// TIA Portal V17 export
// export: Created 2025-07-01T09:58:25.4469357Z, ExportSetting WithDefaults, DisplayName Totally Integrated Automation Portal, DisplayVersion V17 Update 8, DisplayName TIA Portal Openness, DisplayVersion V17 Update 8, DisplayName TIA Portal Version Control Interface, DisplayVersion V17, DisplayName SINAMICS Startdrive Advanced, DisplayVersion V17 SP2, DisplayName SINAMICS Startdrive G110M, G120, G120C, G120D, G120P, G115D, DisplayVersion V17 SP2, DisplayName SINAMICS Startdrive G130, G150, S120, S150, SINAMICS MV, S210, DisplayVersion V17 SP2, DisplayName STEP 7 Professional, DisplayVersion V17 Update 8, DisplayName SINUMERIK ONE STEP 7 Toolbox, DisplayVersion V17 Update 12, DisplayName SINUMERIK ONE PLC Basic Program Plus, DisplayVersion V17 Update 12, DisplayName SINUMERIK 840D sl STEP 7 Toolbox, DisplayVersion V17 Update 12, DisplayName STEP 7 Safety, DisplayVersion V17 Update 6, DisplayName WinCC Advanced, DisplayVersion V17 Update 8
FUNCTION "FC2500_UNIT_1_FIXTURES" : Void   // FC2500, LAD
TITLE = FIXTURE 1
{ S7_Optimized_Access := 'FALSE' }
AUTHOR : ETXETAR
VERSION : 1.0
// stored: AutoNumber false, IsIECCheckEnabled false, SetENOAutomatically false, UDAEnableTagReadback false
   VAR CONSTANT
      FC_NUMBER : DInt := 2500;
   END_VAR
BEGIN

REGION Network 1: CALL FB2500 FIXTURE 1 UNIT 1 CLADDING
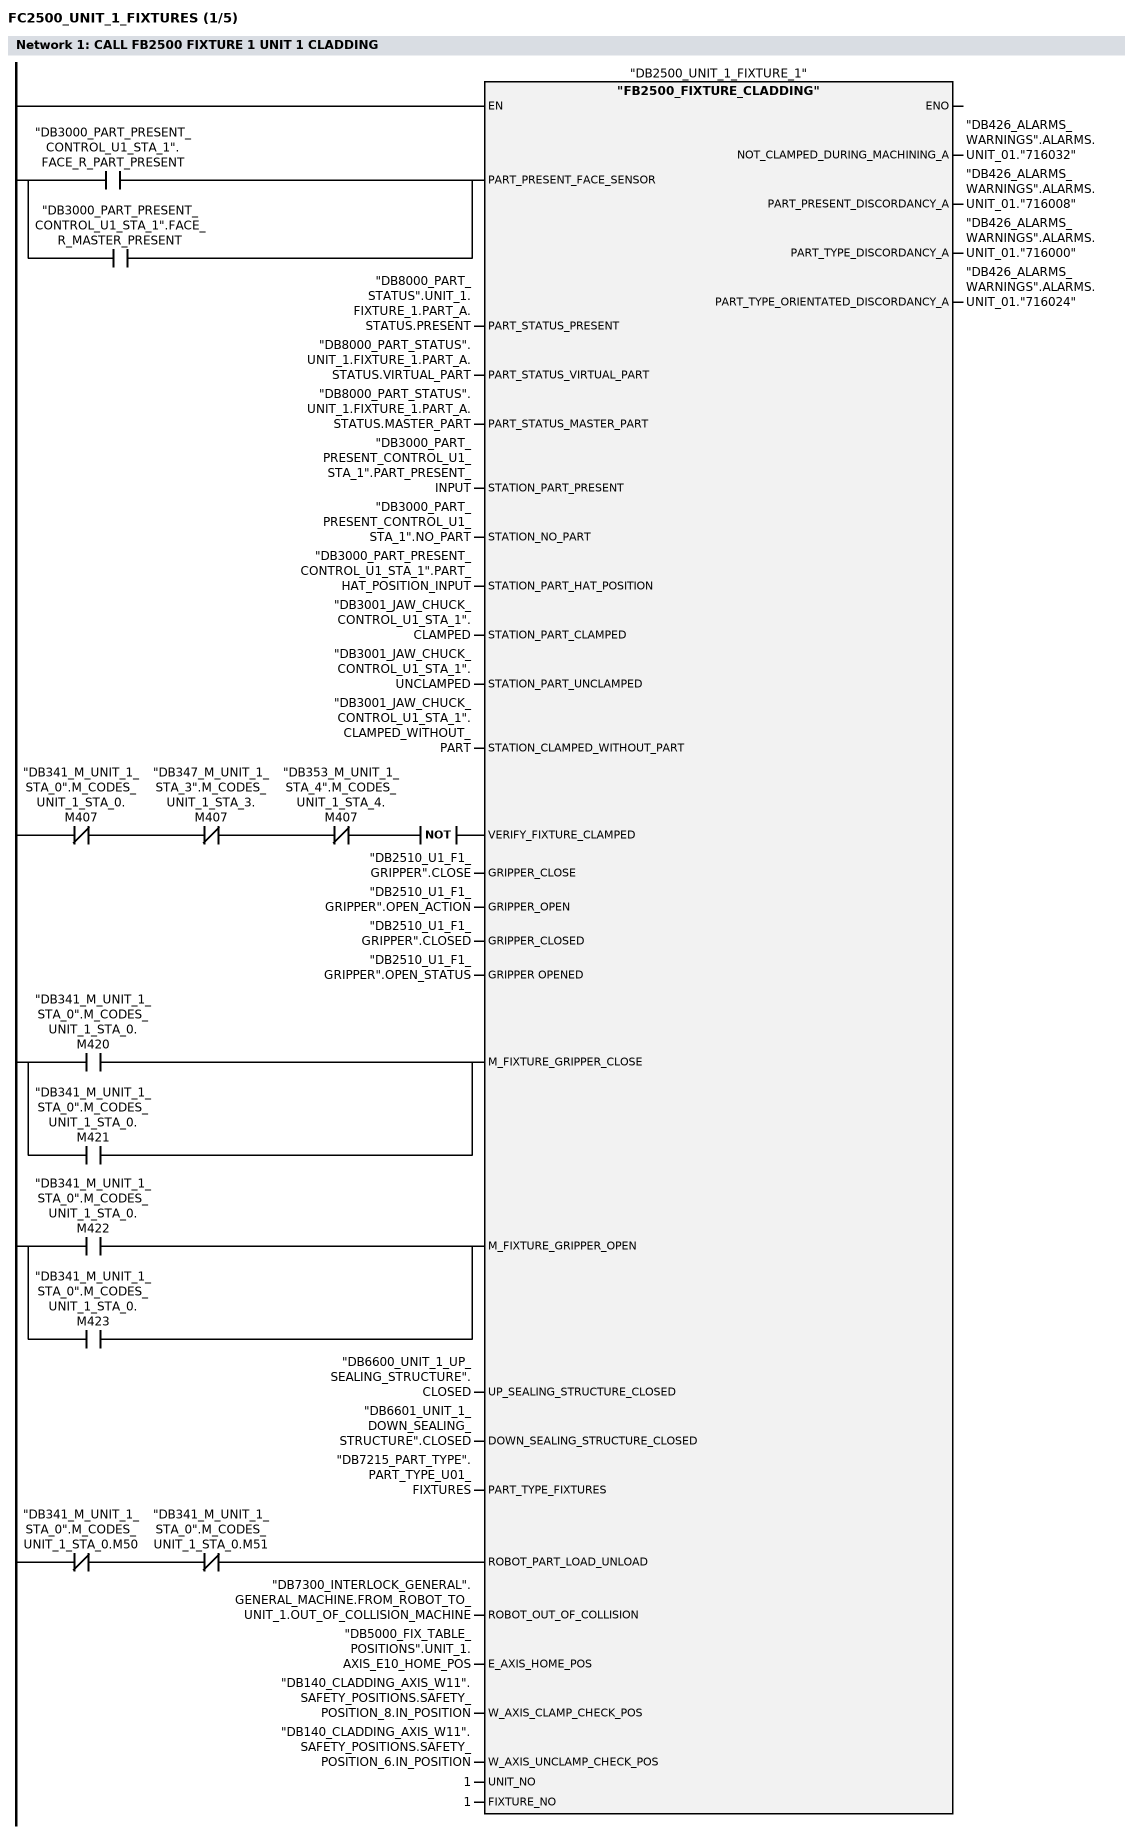
   RUNG wire#powerrail
      "DB2500_UNIT_1_FIXTURE_1"(PART_PRESENT_FACE_SENSOR := wire#w1, VERIFY_FIXTURE_CLAMPED := wire#w2, M_FIXTURE_GRIPPER_CLOSE := wire#w3, M_FIXTURE_GRIPPER_OPEN := wire#w4, ROBOT_PART_LOAD_UNLOAD := wire#w5, PART_STATUS_PRESENT := "DB8000_PART_STATUS".UNIT_1.FIXTURE_1.PART_A.STATUS.PRESENT, PART_STATUS_VIRTUAL_PART := "DB8000_PART_STATUS".UNIT_1.FIXTURE_1.PART_A.STATUS.VIRTUAL_PART, PART_STATUS_MASTER_PART := "DB8000_PART_STATUS".UNIT_1.FIXTURE_1.PART_A.STATUS.MASTER_PART, STATION_PART_PRESENT := "DB3000_PART_PRESENT_CONTROL_U1_STA_1".PART_PRESENT_INPUT, STATION_NO_PART := "DB3000_PART_PRESENT_CONTROL_U1_STA_1".NO_PART, STATION_PART_HAT_POSITION := "DB3000_PART_PRESENT_CONTROL_U1_STA_1".PART_HAT_POSITION_INPUT, STATION_PART_CLAMPED := "DB3001_JAW_CHUCK_CONTROL_U1_STA_1".CLAMPED, STATION_PART_UNCLAMPED := "DB3001_JAW_CHUCK_CONTROL_U1_STA_1".UNCLAMPED, STATION_CLAMPED_WITHOUT_PART := "DB3001_JAW_CHUCK_CONTROL_U1_STA_1".CLAMPED_WITHOUT_PART, GRIPPER_CLOSE := "DB2510_U1_F1_GRIPPER".CLOSE, GRIPPER_OPEN := "DB2510_U1_F1_GRIPPER".OPEN_ACTION, GRIPPER_CLOSED := "DB2510_U1_F1_GRIPPER".CLOSED, "GRIPPER OPENED" := "DB2510_U1_F1_GRIPPER".OPEN_STATUS, UP_SEALING_STRUCTURE_CLOSED := "DB6600_UNIT_1_UP_SEALING_STRUCTURE".CLOSED, DOWN_SEALING_STRUCTURE_CLOSED := "DB6601_UNIT_1_DOWN_SEALING_STRUCTURE".CLOSED, PART_TYPE_FIXTURES := "DB7215_PART_TYPE".PART_TYPE_U01_FIXTURES, ROBOT_OUT_OF_COLLISION := "DB7300_INTERLOCK_GENERAL".GENERAL_MACHINE.FROM_ROBOT_TO_UNIT_1.OUT_OF_COLLISION_MACHINE, E_AXIS_HOME_POS := "DB5000_FIX_TABLE_POSITIONS".UNIT_1.AXIS_E10_HOME_POS, W_AXIS_CLAMP_CHECK_POS := "DB140_CLADDING_AXIS_W11".SAFETY_POSITIONS.SAFETY_POSITION_8.IN_POSITION, W_AXIS_UNCLAMP_CHECK_POS := "DB140_CLADDING_AXIS_W11".SAFETY_POSITIONS.SAFETY_POSITION_6.IN_POSITION, UNIT_NO := 1, FIXTURE_NO := 1, NOT_CLAMPED_DURING_MACHINING_A => "DB426_ALARMS_WARNINGS".ALARMS.UNIT_01."716032", PART_PRESENT_DISCORDANCY_A => "DB426_ALARMS_WARNINGS".ALARMS.UNIT_01."716008", PART_TYPE_DISCORDANCY_A => "DB426_ALARMS_WARNINGS".ALARMS.UNIT_01."716000", PART_TYPE_ORIENTATED_DISCORDANCY_A => "DB426_ALARMS_WARNINGS".ALARMS.UNIT_01."716024")
   END_RUNG
   RUNG wire#powerrail
      Contact( "DB3000_PART_PRESENT_CONTROL_U1_STA_1".FACE_R_PART_PRESENT )
   END_RUNG wire#w1
   RUNG wire#powerrail
      Contact( "DB3000_PART_PRESENT_CONTROL_U1_STA_1".FACE_R_MASTER_PRESENT )
   END_RUNG wire#w1
   RUNG wire#powerrail
      I_Contact( "DB341_M_UNIT_1_STA_0".M_CODES_UNIT_1_STA_0.M407 )
      I_Contact( "DB347_M_UNIT_1_STA_3".M_CODES_UNIT_1_STA_3.M407 )
      I_Contact( "DB353_M_UNIT_1_STA_4".M_CODES_UNIT_1_STA_4.M407 )
      Not()
   END_RUNG wire#w2
   RUNG wire#powerrail
      Contact( "DB341_M_UNIT_1_STA_0".M_CODES_UNIT_1_STA_0.M420 )
   END_RUNG wire#w3
   RUNG wire#powerrail
      Contact( "DB341_M_UNIT_1_STA_0".M_CODES_UNIT_1_STA_0.M421 )
   END_RUNG wire#w3
   RUNG wire#powerrail
      Contact( "DB341_M_UNIT_1_STA_0".M_CODES_UNIT_1_STA_0.M422 )
   END_RUNG wire#w4
   RUNG wire#powerrail
      Contact( "DB341_M_UNIT_1_STA_0".M_CODES_UNIT_1_STA_0.M423 )
   END_RUNG wire#w4
   RUNG wire#powerrail
      I_Contact( "DB341_M_UNIT_1_STA_0".M_CODES_UNIT_1_STA_0.M50 )
      I_Contact( "DB341_M_UNIT_1_STA_0".M_CODES_UNIT_1_STA_0.M51 )
   END_RUNG wire#w5
   // the same network as SCL:
   "DB2500_UNIT_1_FIXTURE_1"(PART_PRESENT_FACE_SENSOR := "DB3000_PART_PRESENT_CONTROL_U1_STA_1".FACE_R_PART_PRESENT OR "DB3000_PART_PRESENT_CONTROL_U1_STA_1".FACE_R_MASTER_PRESENT,   // "FB2500_FIXTURE_CLADDING"
                           PART_STATUS_PRESENT := "DB8000_PART_STATUS".UNIT_1.FIXTURE_1.PART_A.STATUS.PRESENT,
                           PART_STATUS_VIRTUAL_PART := "DB8000_PART_STATUS".UNIT_1.FIXTURE_1.PART_A.STATUS.VIRTUAL_PART,
                           PART_STATUS_MASTER_PART := "DB8000_PART_STATUS".UNIT_1.FIXTURE_1.PART_A.STATUS.MASTER_PART,
                           STATION_PART_PRESENT := "DB3000_PART_PRESENT_CONTROL_U1_STA_1".PART_PRESENT_INPUT,
                           STATION_NO_PART := "DB3000_PART_PRESENT_CONTROL_U1_STA_1".NO_PART,
                           STATION_PART_HAT_POSITION := "DB3000_PART_PRESENT_CONTROL_U1_STA_1".PART_HAT_POSITION_INPUT,
                           STATION_PART_CLAMPED := "DB3001_JAW_CHUCK_CONTROL_U1_STA_1".CLAMPED,
                           STATION_PART_UNCLAMPED := "DB3001_JAW_CHUCK_CONTROL_U1_STA_1".UNCLAMPED,
                           STATION_CLAMPED_WITHOUT_PART := "DB3001_JAW_CHUCK_CONTROL_U1_STA_1".CLAMPED_WITHOUT_PART,
                           VERIFY_FIXTURE_CLAMPED := NOT (NOT "DB341_M_UNIT_1_STA_0".M_CODES_UNIT_1_STA_0.M407 AND NOT "DB347_M_UNIT_1_STA_3".M_CODES_UNIT_1_STA_3.M407 AND NOT "DB353_M_UNIT_1_STA_4".M_CODES_UNIT_1_STA_4.M407),
                           GRIPPER_CLOSE := "DB2510_U1_F1_GRIPPER".CLOSE,
                           GRIPPER_OPEN := "DB2510_U1_F1_GRIPPER".OPEN_ACTION,
                           GRIPPER_CLOSED := "DB2510_U1_F1_GRIPPER".CLOSED,
                           "GRIPPER OPENED" := "DB2510_U1_F1_GRIPPER".OPEN_STATUS,
                           M_FIXTURE_GRIPPER_CLOSE := "DB341_M_UNIT_1_STA_0".M_CODES_UNIT_1_STA_0.M420 OR "DB341_M_UNIT_1_STA_0".M_CODES_UNIT_1_STA_0.M421,
                           M_FIXTURE_GRIPPER_OPEN := "DB341_M_UNIT_1_STA_0".M_CODES_UNIT_1_STA_0.M422 OR "DB341_M_UNIT_1_STA_0".M_CODES_UNIT_1_STA_0.M423,
                           UP_SEALING_STRUCTURE_CLOSED := "DB6600_UNIT_1_UP_SEALING_STRUCTURE".CLOSED,
                           DOWN_SEALING_STRUCTURE_CLOSED := "DB6601_UNIT_1_DOWN_SEALING_STRUCTURE".CLOSED,
                           PART_TYPE_FIXTURES := "DB7215_PART_TYPE".PART_TYPE_U01_FIXTURES,
                           ROBOT_PART_LOAD_UNLOAD := NOT "DB341_M_UNIT_1_STA_0".M_CODES_UNIT_1_STA_0.M50 AND NOT "DB341_M_UNIT_1_STA_0".M_CODES_UNIT_1_STA_0.M51,
                           ROBOT_OUT_OF_COLLISION := "DB7300_INTERLOCK_GENERAL".GENERAL_MACHINE.FROM_ROBOT_TO_UNIT_1.OUT_OF_COLLISION_MACHINE,
                           E_AXIS_HOME_POS := "DB5000_FIX_TABLE_POSITIONS".UNIT_1.AXIS_E10_HOME_POS,
                           W_AXIS_CLAMP_CHECK_POS := "DB140_CLADDING_AXIS_W11".SAFETY_POSITIONS.SAFETY_POSITION_8.IN_POSITION,
                           W_AXIS_UNCLAMP_CHECK_POS := "DB140_CLADDING_AXIS_W11".SAFETY_POSITIONS.SAFETY_POSITION_6.IN_POSITION,
                           UNIT_NO := 1,
                           FIXTURE_NO := 1,
                           NOT_CLAMPED_DURING_MACHINING_A => "DB426_ALARMS_WARNINGS".ALARMS.UNIT_01."716032",
                           PART_PRESENT_DISCORDANCY_A => "DB426_ALARMS_WARNINGS".ALARMS.UNIT_01."716008",
                           PART_TYPE_DISCORDANCY_A => "DB426_ALARMS_WARNINGS".ALARMS.UNIT_01."716000",
                           PART_TYPE_ORIENTATED_DISCORDANCY_A => "DB426_ALARMS_WARNINGS".ALARMS.UNIT_01."716024");
END_REGION

REGION Network 2: CALL FB2600 FIXTURE 2 UNIT 1 CLADDING
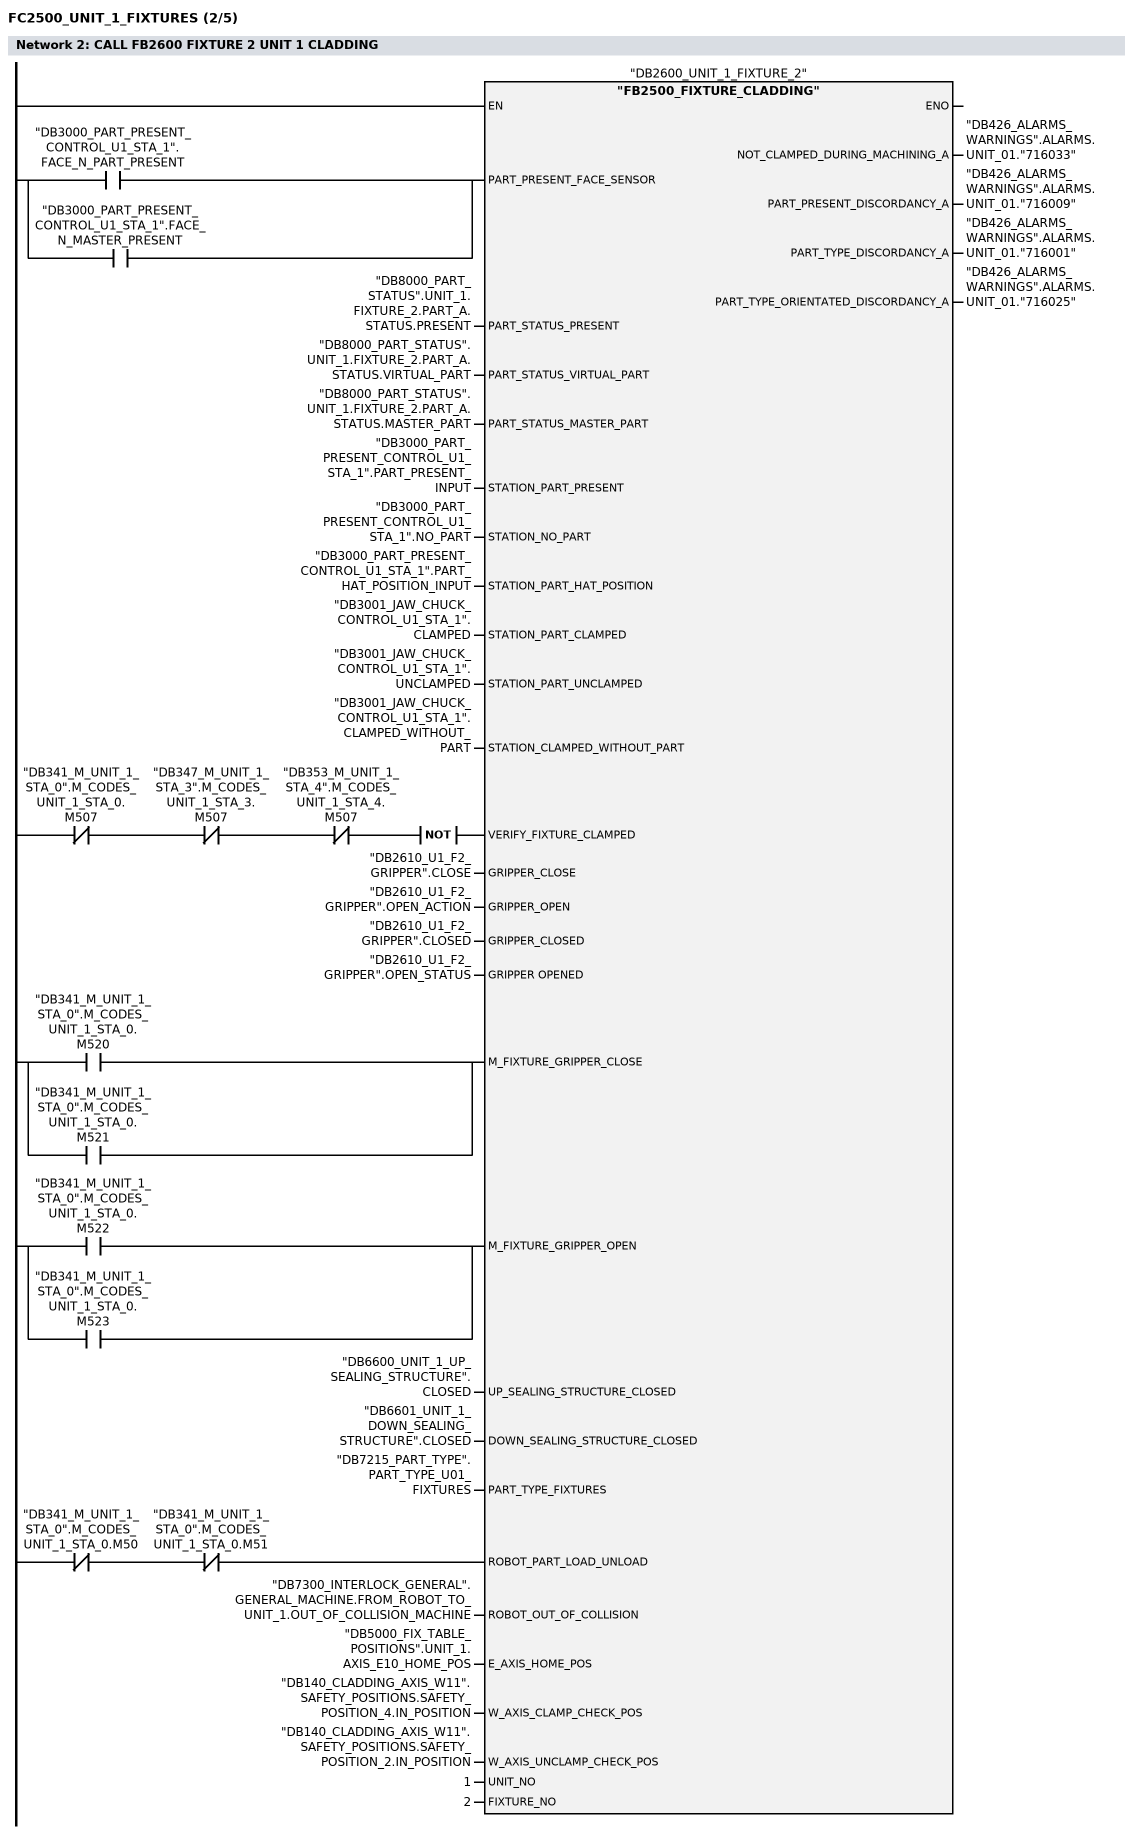
   RUNG wire#powerrail
      "DB2600_UNIT_1_FIXTURE_2"(PART_PRESENT_FACE_SENSOR := wire#w1, VERIFY_FIXTURE_CLAMPED := wire#w2, M_FIXTURE_GRIPPER_CLOSE := wire#w3, M_FIXTURE_GRIPPER_OPEN := wire#w4, ROBOT_PART_LOAD_UNLOAD := wire#w5, PART_STATUS_PRESENT := "DB8000_PART_STATUS".UNIT_1.FIXTURE_2.PART_A.STATUS.PRESENT, PART_STATUS_VIRTUAL_PART := "DB8000_PART_STATUS".UNIT_1.FIXTURE_2.PART_A.STATUS.VIRTUAL_PART, PART_STATUS_MASTER_PART := "DB8000_PART_STATUS".UNIT_1.FIXTURE_2.PART_A.STATUS.MASTER_PART, STATION_PART_PRESENT := "DB3000_PART_PRESENT_CONTROL_U1_STA_1".PART_PRESENT_INPUT, STATION_NO_PART := "DB3000_PART_PRESENT_CONTROL_U1_STA_1".NO_PART, STATION_PART_HAT_POSITION := "DB3000_PART_PRESENT_CONTROL_U1_STA_1".PART_HAT_POSITION_INPUT, STATION_PART_CLAMPED := "DB3001_JAW_CHUCK_CONTROL_U1_STA_1".CLAMPED, STATION_PART_UNCLAMPED := "DB3001_JAW_CHUCK_CONTROL_U1_STA_1".UNCLAMPED, STATION_CLAMPED_WITHOUT_PART := "DB3001_JAW_CHUCK_CONTROL_U1_STA_1".CLAMPED_WITHOUT_PART, GRIPPER_CLOSE := "DB2610_U1_F2_GRIPPER".CLOSE, GRIPPER_OPEN := "DB2610_U1_F2_GRIPPER".OPEN_ACTION, GRIPPER_CLOSED := "DB2610_U1_F2_GRIPPER".CLOSED, "GRIPPER OPENED" := "DB2610_U1_F2_GRIPPER".OPEN_STATUS, UP_SEALING_STRUCTURE_CLOSED := "DB6600_UNIT_1_UP_SEALING_STRUCTURE".CLOSED, DOWN_SEALING_STRUCTURE_CLOSED := "DB6601_UNIT_1_DOWN_SEALING_STRUCTURE".CLOSED, PART_TYPE_FIXTURES := "DB7215_PART_TYPE".PART_TYPE_U01_FIXTURES, ROBOT_OUT_OF_COLLISION := "DB7300_INTERLOCK_GENERAL".GENERAL_MACHINE.FROM_ROBOT_TO_UNIT_1.OUT_OF_COLLISION_MACHINE, E_AXIS_HOME_POS := "DB5000_FIX_TABLE_POSITIONS".UNIT_1.AXIS_E10_HOME_POS, W_AXIS_CLAMP_CHECK_POS := "DB140_CLADDING_AXIS_W11".SAFETY_POSITIONS.SAFETY_POSITION_4.IN_POSITION, W_AXIS_UNCLAMP_CHECK_POS := "DB140_CLADDING_AXIS_W11".SAFETY_POSITIONS.SAFETY_POSITION_2.IN_POSITION, UNIT_NO := 1, FIXTURE_NO := 2, NOT_CLAMPED_DURING_MACHINING_A => "DB426_ALARMS_WARNINGS".ALARMS.UNIT_01."716033", PART_PRESENT_DISCORDANCY_A => "DB426_ALARMS_WARNINGS".ALARMS.UNIT_01."716009", PART_TYPE_DISCORDANCY_A => "DB426_ALARMS_WARNINGS".ALARMS.UNIT_01."716001", PART_TYPE_ORIENTATED_DISCORDANCY_A => "DB426_ALARMS_WARNINGS".ALARMS.UNIT_01."716025")
   END_RUNG
   RUNG wire#powerrail
      Contact( "DB3000_PART_PRESENT_CONTROL_U1_STA_1".FACE_N_PART_PRESENT )
   END_RUNG wire#w1
   RUNG wire#powerrail
      Contact( "DB3000_PART_PRESENT_CONTROL_U1_STA_1".FACE_N_MASTER_PRESENT )
   END_RUNG wire#w1
   RUNG wire#powerrail
      I_Contact( "DB341_M_UNIT_1_STA_0".M_CODES_UNIT_1_STA_0.M507 )
      I_Contact( "DB347_M_UNIT_1_STA_3".M_CODES_UNIT_1_STA_3.M507 )
      I_Contact( "DB353_M_UNIT_1_STA_4".M_CODES_UNIT_1_STA_4.M507 )
      Not()
   END_RUNG wire#w2
   RUNG wire#powerrail
      Contact( "DB341_M_UNIT_1_STA_0".M_CODES_UNIT_1_STA_0.M520 )
   END_RUNG wire#w3
   RUNG wire#powerrail
      Contact( "DB341_M_UNIT_1_STA_0".M_CODES_UNIT_1_STA_0.M521 )
   END_RUNG wire#w3
   RUNG wire#powerrail
      Contact( "DB341_M_UNIT_1_STA_0".M_CODES_UNIT_1_STA_0.M522 )
   END_RUNG wire#w4
   RUNG wire#powerrail
      Contact( "DB341_M_UNIT_1_STA_0".M_CODES_UNIT_1_STA_0.M523 )
   END_RUNG wire#w4
   RUNG wire#powerrail
      I_Contact( "DB341_M_UNIT_1_STA_0".M_CODES_UNIT_1_STA_0.M50 )
      I_Contact( "DB341_M_UNIT_1_STA_0".M_CODES_UNIT_1_STA_0.M51 )
   END_RUNG wire#w5
   // the same network as SCL:
   "DB2600_UNIT_1_FIXTURE_2"(PART_PRESENT_FACE_SENSOR := "DB3000_PART_PRESENT_CONTROL_U1_STA_1".FACE_N_PART_PRESENT OR "DB3000_PART_PRESENT_CONTROL_U1_STA_1".FACE_N_MASTER_PRESENT,   // "FB2500_FIXTURE_CLADDING"
                           PART_STATUS_PRESENT := "DB8000_PART_STATUS".UNIT_1.FIXTURE_2.PART_A.STATUS.PRESENT,
                           PART_STATUS_VIRTUAL_PART := "DB8000_PART_STATUS".UNIT_1.FIXTURE_2.PART_A.STATUS.VIRTUAL_PART,
                           PART_STATUS_MASTER_PART := "DB8000_PART_STATUS".UNIT_1.FIXTURE_2.PART_A.STATUS.MASTER_PART,
                           STATION_PART_PRESENT := "DB3000_PART_PRESENT_CONTROL_U1_STA_1".PART_PRESENT_INPUT,
                           STATION_NO_PART := "DB3000_PART_PRESENT_CONTROL_U1_STA_1".NO_PART,
                           STATION_PART_HAT_POSITION := "DB3000_PART_PRESENT_CONTROL_U1_STA_1".PART_HAT_POSITION_INPUT,
                           STATION_PART_CLAMPED := "DB3001_JAW_CHUCK_CONTROL_U1_STA_1".CLAMPED,
                           STATION_PART_UNCLAMPED := "DB3001_JAW_CHUCK_CONTROL_U1_STA_1".UNCLAMPED,
                           STATION_CLAMPED_WITHOUT_PART := "DB3001_JAW_CHUCK_CONTROL_U1_STA_1".CLAMPED_WITHOUT_PART,
                           VERIFY_FIXTURE_CLAMPED := NOT (NOT "DB341_M_UNIT_1_STA_0".M_CODES_UNIT_1_STA_0.M507 AND NOT "DB347_M_UNIT_1_STA_3".M_CODES_UNIT_1_STA_3.M507 AND NOT "DB353_M_UNIT_1_STA_4".M_CODES_UNIT_1_STA_4.M507),
                           GRIPPER_CLOSE := "DB2610_U1_F2_GRIPPER".CLOSE,
                           GRIPPER_OPEN := "DB2610_U1_F2_GRIPPER".OPEN_ACTION,
                           GRIPPER_CLOSED := "DB2610_U1_F2_GRIPPER".CLOSED,
                           "GRIPPER OPENED" := "DB2610_U1_F2_GRIPPER".OPEN_STATUS,
                           M_FIXTURE_GRIPPER_CLOSE := "DB341_M_UNIT_1_STA_0".M_CODES_UNIT_1_STA_0.M520 OR "DB341_M_UNIT_1_STA_0".M_CODES_UNIT_1_STA_0.M521,
                           M_FIXTURE_GRIPPER_OPEN := "DB341_M_UNIT_1_STA_0".M_CODES_UNIT_1_STA_0.M522 OR "DB341_M_UNIT_1_STA_0".M_CODES_UNIT_1_STA_0.M523,
                           UP_SEALING_STRUCTURE_CLOSED := "DB6600_UNIT_1_UP_SEALING_STRUCTURE".CLOSED,
                           DOWN_SEALING_STRUCTURE_CLOSED := "DB6601_UNIT_1_DOWN_SEALING_STRUCTURE".CLOSED,
                           PART_TYPE_FIXTURES := "DB7215_PART_TYPE".PART_TYPE_U01_FIXTURES,
                           ROBOT_PART_LOAD_UNLOAD := NOT "DB341_M_UNIT_1_STA_0".M_CODES_UNIT_1_STA_0.M50 AND NOT "DB341_M_UNIT_1_STA_0".M_CODES_UNIT_1_STA_0.M51,
                           ROBOT_OUT_OF_COLLISION := "DB7300_INTERLOCK_GENERAL".GENERAL_MACHINE.FROM_ROBOT_TO_UNIT_1.OUT_OF_COLLISION_MACHINE,
                           E_AXIS_HOME_POS := "DB5000_FIX_TABLE_POSITIONS".UNIT_1.AXIS_E10_HOME_POS,
                           W_AXIS_CLAMP_CHECK_POS := "DB140_CLADDING_AXIS_W11".SAFETY_POSITIONS.SAFETY_POSITION_4.IN_POSITION,
                           W_AXIS_UNCLAMP_CHECK_POS := "DB140_CLADDING_AXIS_W11".SAFETY_POSITIONS.SAFETY_POSITION_2.IN_POSITION,
                           UNIT_NO := 1,
                           FIXTURE_NO := 2,
                           NOT_CLAMPED_DURING_MACHINING_A => "DB426_ALARMS_WARNINGS".ALARMS.UNIT_01."716033",
                           PART_PRESENT_DISCORDANCY_A => "DB426_ALARMS_WARNINGS".ALARMS.UNIT_01."716009",
                           PART_TYPE_DISCORDANCY_A => "DB426_ALARMS_WARNINGS".ALARMS.UNIT_01."716001",
                           PART_TYPE_ORIENTATED_DISCORDANCY_A => "DB426_ALARMS_WARNINGS".ALARMS.UNIT_01."716025");
END_REGION

REGION Network 3: CALL FB2600 FIXTURE 3 UNIT 1 CLADDING
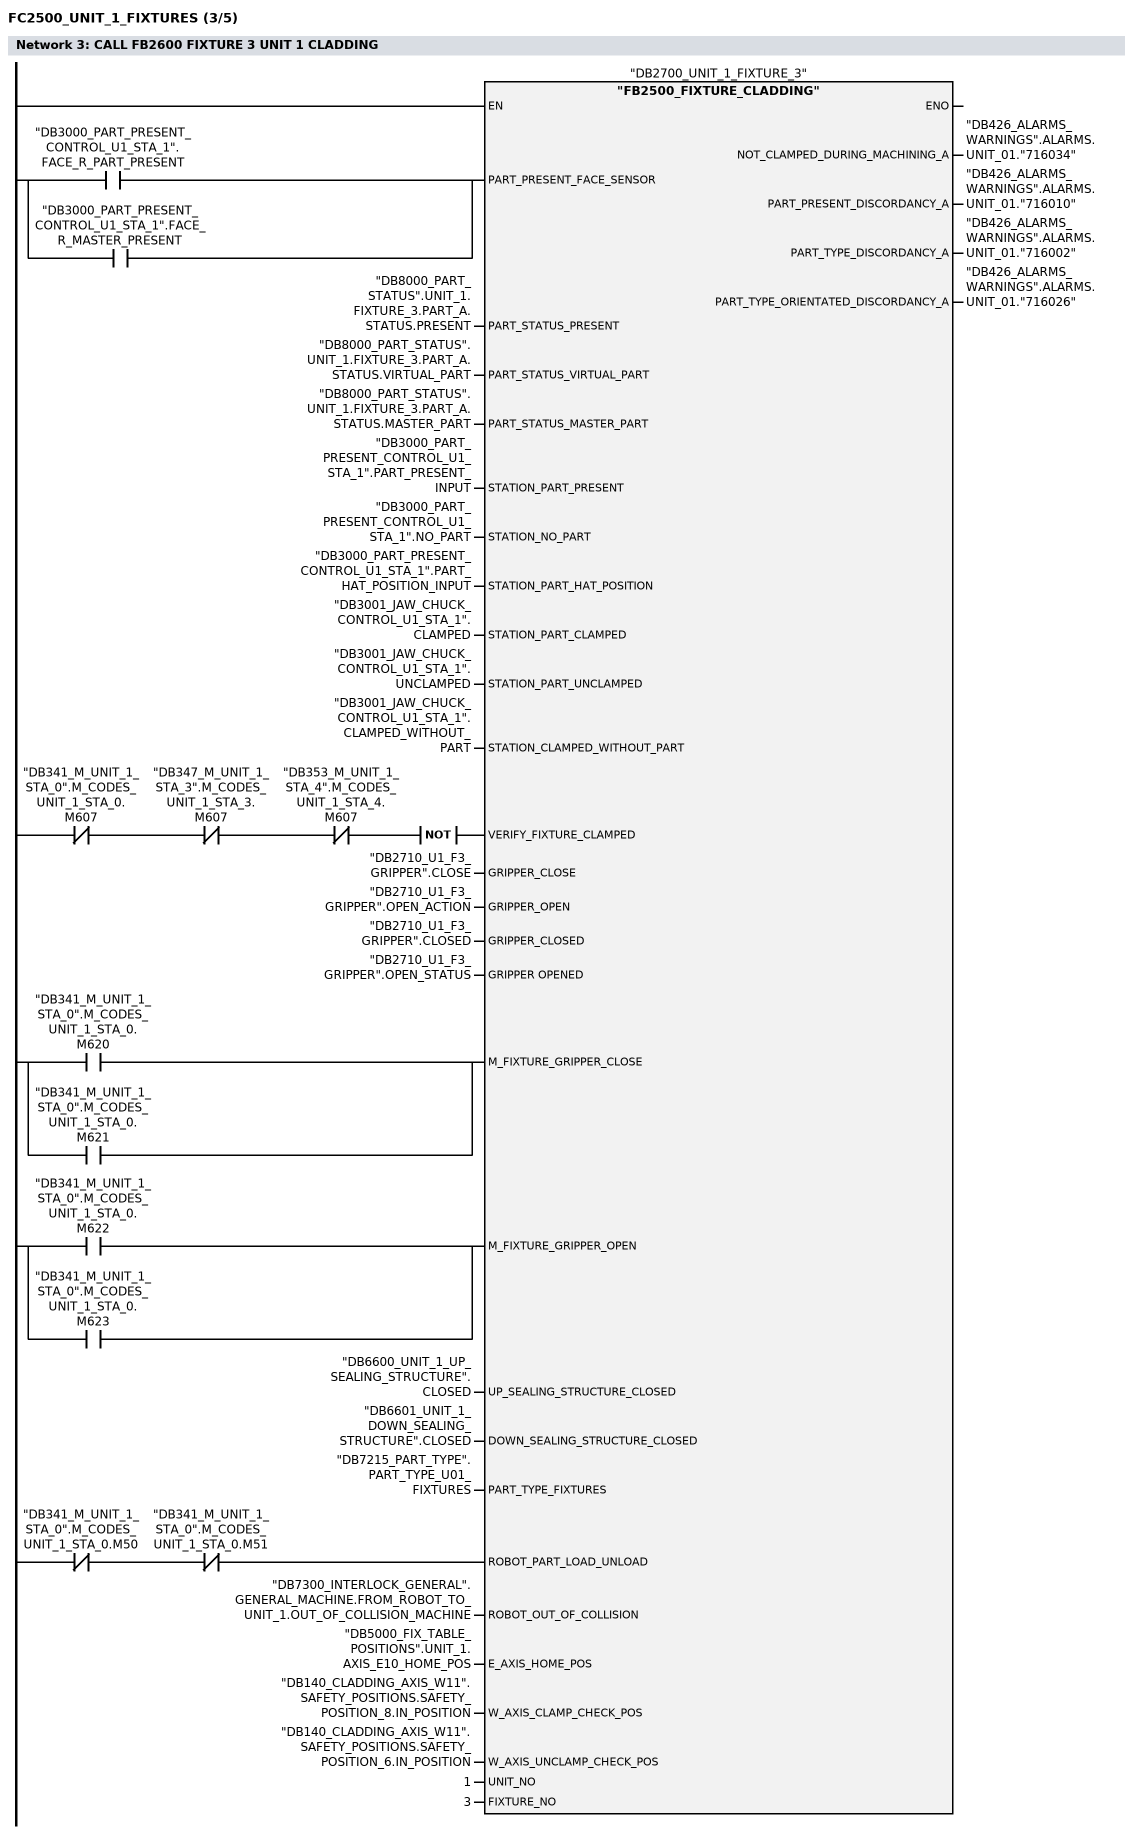
   RUNG wire#powerrail
      "DB2700_UNIT_1_FIXTURE_3"(PART_PRESENT_FACE_SENSOR := wire#w1, VERIFY_FIXTURE_CLAMPED := wire#w2, M_FIXTURE_GRIPPER_CLOSE := wire#w3, M_FIXTURE_GRIPPER_OPEN := wire#w4, ROBOT_PART_LOAD_UNLOAD := wire#w5, PART_STATUS_PRESENT := "DB8000_PART_STATUS".UNIT_1.FIXTURE_3.PART_A.STATUS.PRESENT, PART_STATUS_VIRTUAL_PART := "DB8000_PART_STATUS".UNIT_1.FIXTURE_3.PART_A.STATUS.VIRTUAL_PART, PART_STATUS_MASTER_PART := "DB8000_PART_STATUS".UNIT_1.FIXTURE_3.PART_A.STATUS.MASTER_PART, STATION_PART_PRESENT := "DB3000_PART_PRESENT_CONTROL_U1_STA_1".PART_PRESENT_INPUT, STATION_NO_PART := "DB3000_PART_PRESENT_CONTROL_U1_STA_1".NO_PART, STATION_PART_HAT_POSITION := "DB3000_PART_PRESENT_CONTROL_U1_STA_1".PART_HAT_POSITION_INPUT, STATION_PART_CLAMPED := "DB3001_JAW_CHUCK_CONTROL_U1_STA_1".CLAMPED, STATION_PART_UNCLAMPED := "DB3001_JAW_CHUCK_CONTROL_U1_STA_1".UNCLAMPED, STATION_CLAMPED_WITHOUT_PART := "DB3001_JAW_CHUCK_CONTROL_U1_STA_1".CLAMPED_WITHOUT_PART, GRIPPER_CLOSE := "DB2710_U1_F3_GRIPPER".CLOSE, GRIPPER_OPEN := "DB2710_U1_F3_GRIPPER".OPEN_ACTION, GRIPPER_CLOSED := "DB2710_U1_F3_GRIPPER".CLOSED, "GRIPPER OPENED" := "DB2710_U1_F3_GRIPPER".OPEN_STATUS, UP_SEALING_STRUCTURE_CLOSED := "DB6600_UNIT_1_UP_SEALING_STRUCTURE".CLOSED, DOWN_SEALING_STRUCTURE_CLOSED := "DB6601_UNIT_1_DOWN_SEALING_STRUCTURE".CLOSED, PART_TYPE_FIXTURES := "DB7215_PART_TYPE".PART_TYPE_U01_FIXTURES, ROBOT_OUT_OF_COLLISION := "DB7300_INTERLOCK_GENERAL".GENERAL_MACHINE.FROM_ROBOT_TO_UNIT_1.OUT_OF_COLLISION_MACHINE, E_AXIS_HOME_POS := "DB5000_FIX_TABLE_POSITIONS".UNIT_1.AXIS_E10_HOME_POS, W_AXIS_CLAMP_CHECK_POS := "DB140_CLADDING_AXIS_W11".SAFETY_POSITIONS.SAFETY_POSITION_8.IN_POSITION, W_AXIS_UNCLAMP_CHECK_POS := "DB140_CLADDING_AXIS_W11".SAFETY_POSITIONS.SAFETY_POSITION_6.IN_POSITION, UNIT_NO := 1, FIXTURE_NO := 3, NOT_CLAMPED_DURING_MACHINING_A => "DB426_ALARMS_WARNINGS".ALARMS.UNIT_01."716034", PART_PRESENT_DISCORDANCY_A => "DB426_ALARMS_WARNINGS".ALARMS.UNIT_01."716010", PART_TYPE_DISCORDANCY_A => "DB426_ALARMS_WARNINGS".ALARMS.UNIT_01."716002", PART_TYPE_ORIENTATED_DISCORDANCY_A => "DB426_ALARMS_WARNINGS".ALARMS.UNIT_01."716026")
   END_RUNG
   RUNG wire#powerrail
      Contact( "DB3000_PART_PRESENT_CONTROL_U1_STA_1".FACE_R_PART_PRESENT )
   END_RUNG wire#w1
   RUNG wire#powerrail
      Contact( "DB3000_PART_PRESENT_CONTROL_U1_STA_1".FACE_R_MASTER_PRESENT )
   END_RUNG wire#w1
   RUNG wire#powerrail
      I_Contact( "DB341_M_UNIT_1_STA_0".M_CODES_UNIT_1_STA_0.M607 )
      I_Contact( "DB347_M_UNIT_1_STA_3".M_CODES_UNIT_1_STA_3.M607 )
      I_Contact( "DB353_M_UNIT_1_STA_4".M_CODES_UNIT_1_STA_4.M607 )
      Not()
   END_RUNG wire#w2
   RUNG wire#powerrail
      Contact( "DB341_M_UNIT_1_STA_0".M_CODES_UNIT_1_STA_0.M620 )
   END_RUNG wire#w3
   RUNG wire#powerrail
      Contact( "DB341_M_UNIT_1_STA_0".M_CODES_UNIT_1_STA_0.M621 )
   END_RUNG wire#w3
   RUNG wire#powerrail
      Contact( "DB341_M_UNIT_1_STA_0".M_CODES_UNIT_1_STA_0.M622 )
   END_RUNG wire#w4
   RUNG wire#powerrail
      Contact( "DB341_M_UNIT_1_STA_0".M_CODES_UNIT_1_STA_0.M623 )
   END_RUNG wire#w4
   RUNG wire#powerrail
      I_Contact( "DB341_M_UNIT_1_STA_0".M_CODES_UNIT_1_STA_0.M50 )
      I_Contact( "DB341_M_UNIT_1_STA_0".M_CODES_UNIT_1_STA_0.M51 )
   END_RUNG wire#w5
   // the same network as SCL:
   "DB2700_UNIT_1_FIXTURE_3"(PART_PRESENT_FACE_SENSOR := "DB3000_PART_PRESENT_CONTROL_U1_STA_1".FACE_R_PART_PRESENT OR "DB3000_PART_PRESENT_CONTROL_U1_STA_1".FACE_R_MASTER_PRESENT,   // "FB2500_FIXTURE_CLADDING"
                           PART_STATUS_PRESENT := "DB8000_PART_STATUS".UNIT_1.FIXTURE_3.PART_A.STATUS.PRESENT,
                           PART_STATUS_VIRTUAL_PART := "DB8000_PART_STATUS".UNIT_1.FIXTURE_3.PART_A.STATUS.VIRTUAL_PART,
                           PART_STATUS_MASTER_PART := "DB8000_PART_STATUS".UNIT_1.FIXTURE_3.PART_A.STATUS.MASTER_PART,
                           STATION_PART_PRESENT := "DB3000_PART_PRESENT_CONTROL_U1_STA_1".PART_PRESENT_INPUT,
                           STATION_NO_PART := "DB3000_PART_PRESENT_CONTROL_U1_STA_1".NO_PART,
                           STATION_PART_HAT_POSITION := "DB3000_PART_PRESENT_CONTROL_U1_STA_1".PART_HAT_POSITION_INPUT,
                           STATION_PART_CLAMPED := "DB3001_JAW_CHUCK_CONTROL_U1_STA_1".CLAMPED,
                           STATION_PART_UNCLAMPED := "DB3001_JAW_CHUCK_CONTROL_U1_STA_1".UNCLAMPED,
                           STATION_CLAMPED_WITHOUT_PART := "DB3001_JAW_CHUCK_CONTROL_U1_STA_1".CLAMPED_WITHOUT_PART,
                           VERIFY_FIXTURE_CLAMPED := NOT (NOT "DB341_M_UNIT_1_STA_0".M_CODES_UNIT_1_STA_0.M607 AND NOT "DB347_M_UNIT_1_STA_3".M_CODES_UNIT_1_STA_3.M607 AND NOT "DB353_M_UNIT_1_STA_4".M_CODES_UNIT_1_STA_4.M607),
                           GRIPPER_CLOSE := "DB2710_U1_F3_GRIPPER".CLOSE,
                           GRIPPER_OPEN := "DB2710_U1_F3_GRIPPER".OPEN_ACTION,
                           GRIPPER_CLOSED := "DB2710_U1_F3_GRIPPER".CLOSED,
                           "GRIPPER OPENED" := "DB2710_U1_F3_GRIPPER".OPEN_STATUS,
                           M_FIXTURE_GRIPPER_CLOSE := "DB341_M_UNIT_1_STA_0".M_CODES_UNIT_1_STA_0.M620 OR "DB341_M_UNIT_1_STA_0".M_CODES_UNIT_1_STA_0.M621,
                           M_FIXTURE_GRIPPER_OPEN := "DB341_M_UNIT_1_STA_0".M_CODES_UNIT_1_STA_0.M622 OR "DB341_M_UNIT_1_STA_0".M_CODES_UNIT_1_STA_0.M623,
                           UP_SEALING_STRUCTURE_CLOSED := "DB6600_UNIT_1_UP_SEALING_STRUCTURE".CLOSED,
                           DOWN_SEALING_STRUCTURE_CLOSED := "DB6601_UNIT_1_DOWN_SEALING_STRUCTURE".CLOSED,
                           PART_TYPE_FIXTURES := "DB7215_PART_TYPE".PART_TYPE_U01_FIXTURES,
                           ROBOT_PART_LOAD_UNLOAD := NOT "DB341_M_UNIT_1_STA_0".M_CODES_UNIT_1_STA_0.M50 AND NOT "DB341_M_UNIT_1_STA_0".M_CODES_UNIT_1_STA_0.M51,
                           ROBOT_OUT_OF_COLLISION := "DB7300_INTERLOCK_GENERAL".GENERAL_MACHINE.FROM_ROBOT_TO_UNIT_1.OUT_OF_COLLISION_MACHINE,
                           E_AXIS_HOME_POS := "DB5000_FIX_TABLE_POSITIONS".UNIT_1.AXIS_E10_HOME_POS,
                           W_AXIS_CLAMP_CHECK_POS := "DB140_CLADDING_AXIS_W11".SAFETY_POSITIONS.SAFETY_POSITION_8.IN_POSITION,
                           W_AXIS_UNCLAMP_CHECK_POS := "DB140_CLADDING_AXIS_W11".SAFETY_POSITIONS.SAFETY_POSITION_6.IN_POSITION,
                           UNIT_NO := 1,
                           FIXTURE_NO := 3,
                           NOT_CLAMPED_DURING_MACHINING_A => "DB426_ALARMS_WARNINGS".ALARMS.UNIT_01."716034",
                           PART_PRESENT_DISCORDANCY_A => "DB426_ALARMS_WARNINGS".ALARMS.UNIT_01."716010",
                           PART_TYPE_DISCORDANCY_A => "DB426_ALARMS_WARNINGS".ALARMS.UNIT_01."716002",
                           PART_TYPE_ORIENTATED_DISCORDANCY_A => "DB426_ALARMS_WARNINGS".ALARMS.UNIT_01."716026");
END_REGION

REGION Network 4: CALL FB2600 FIXTURE 4 UNIT 1 CLADDING
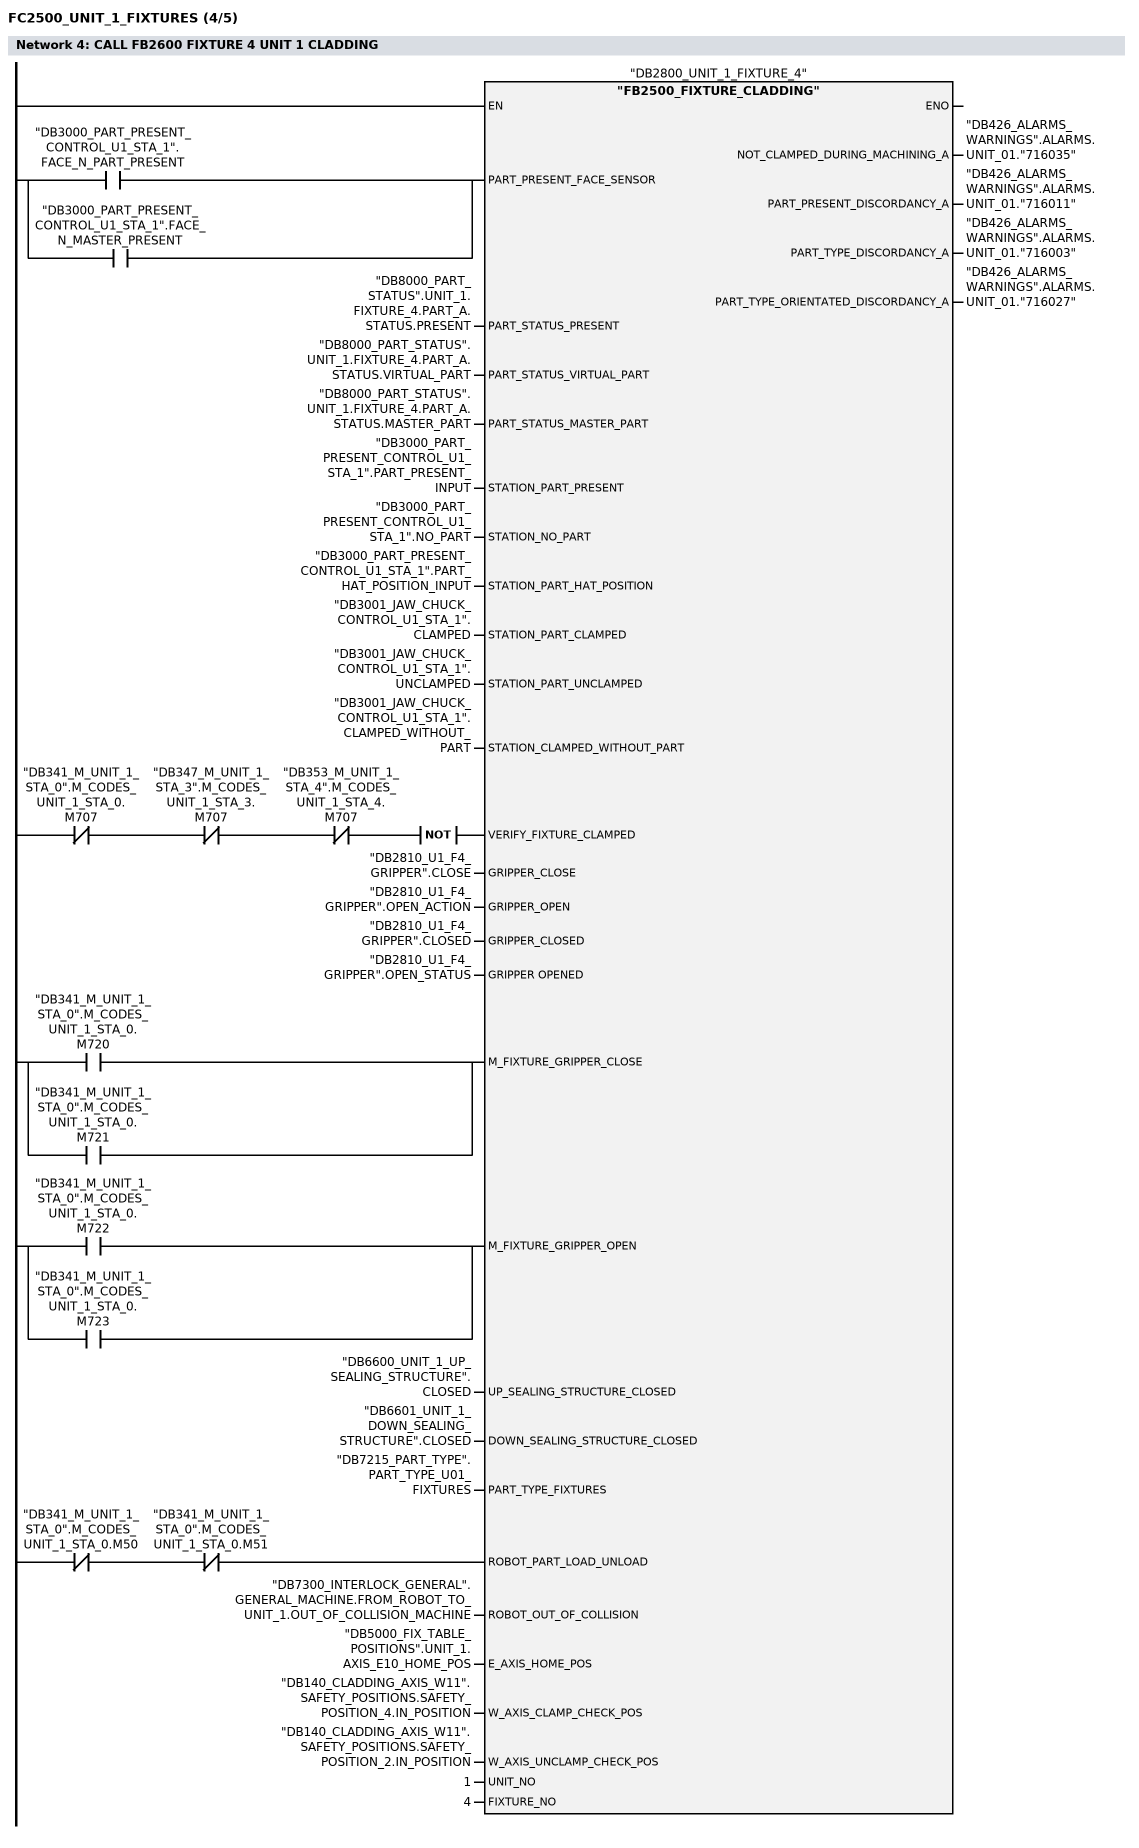
   RUNG wire#powerrail
      "DB2800_UNIT_1_FIXTURE_4"(PART_PRESENT_FACE_SENSOR := wire#w1, VERIFY_FIXTURE_CLAMPED := wire#w2, M_FIXTURE_GRIPPER_CLOSE := wire#w3, M_FIXTURE_GRIPPER_OPEN := wire#w4, ROBOT_PART_LOAD_UNLOAD := wire#w5, PART_STATUS_PRESENT := "DB8000_PART_STATUS".UNIT_1.FIXTURE_4.PART_A.STATUS.PRESENT, PART_STATUS_VIRTUAL_PART := "DB8000_PART_STATUS".UNIT_1.FIXTURE_4.PART_A.STATUS.VIRTUAL_PART, PART_STATUS_MASTER_PART := "DB8000_PART_STATUS".UNIT_1.FIXTURE_4.PART_A.STATUS.MASTER_PART, STATION_PART_PRESENT := "DB3000_PART_PRESENT_CONTROL_U1_STA_1".PART_PRESENT_INPUT, STATION_NO_PART := "DB3000_PART_PRESENT_CONTROL_U1_STA_1".NO_PART, STATION_PART_HAT_POSITION := "DB3000_PART_PRESENT_CONTROL_U1_STA_1".PART_HAT_POSITION_INPUT, STATION_PART_CLAMPED := "DB3001_JAW_CHUCK_CONTROL_U1_STA_1".CLAMPED, STATION_PART_UNCLAMPED := "DB3001_JAW_CHUCK_CONTROL_U1_STA_1".UNCLAMPED, STATION_CLAMPED_WITHOUT_PART := "DB3001_JAW_CHUCK_CONTROL_U1_STA_1".CLAMPED_WITHOUT_PART, GRIPPER_CLOSE := "DB2810_U1_F4_GRIPPER".CLOSE, GRIPPER_OPEN := "DB2810_U1_F4_GRIPPER".OPEN_ACTION, GRIPPER_CLOSED := "DB2810_U1_F4_GRIPPER".CLOSED, "GRIPPER OPENED" := "DB2810_U1_F4_GRIPPER".OPEN_STATUS, UP_SEALING_STRUCTURE_CLOSED := "DB6600_UNIT_1_UP_SEALING_STRUCTURE".CLOSED, DOWN_SEALING_STRUCTURE_CLOSED := "DB6601_UNIT_1_DOWN_SEALING_STRUCTURE".CLOSED, PART_TYPE_FIXTURES := "DB7215_PART_TYPE".PART_TYPE_U01_FIXTURES, ROBOT_OUT_OF_COLLISION := "DB7300_INTERLOCK_GENERAL".GENERAL_MACHINE.FROM_ROBOT_TO_UNIT_1.OUT_OF_COLLISION_MACHINE, E_AXIS_HOME_POS := "DB5000_FIX_TABLE_POSITIONS".UNIT_1.AXIS_E10_HOME_POS, W_AXIS_CLAMP_CHECK_POS := "DB140_CLADDING_AXIS_W11".SAFETY_POSITIONS.SAFETY_POSITION_4.IN_POSITION, W_AXIS_UNCLAMP_CHECK_POS := "DB140_CLADDING_AXIS_W11".SAFETY_POSITIONS.SAFETY_POSITION_2.IN_POSITION, UNIT_NO := 1, FIXTURE_NO := 4, NOT_CLAMPED_DURING_MACHINING_A => "DB426_ALARMS_WARNINGS".ALARMS.UNIT_01."716035", PART_PRESENT_DISCORDANCY_A => "DB426_ALARMS_WARNINGS".ALARMS.UNIT_01."716011", PART_TYPE_DISCORDANCY_A => "DB426_ALARMS_WARNINGS".ALARMS.UNIT_01."716003", PART_TYPE_ORIENTATED_DISCORDANCY_A => "DB426_ALARMS_WARNINGS".ALARMS.UNIT_01."716027")
   END_RUNG
   RUNG wire#powerrail
      Contact( "DB3000_PART_PRESENT_CONTROL_U1_STA_1".FACE_N_PART_PRESENT )
   END_RUNG wire#w1
   RUNG wire#powerrail
      Contact( "DB3000_PART_PRESENT_CONTROL_U1_STA_1".FACE_N_MASTER_PRESENT )
   END_RUNG wire#w1
   RUNG wire#powerrail
      I_Contact( "DB341_M_UNIT_1_STA_0".M_CODES_UNIT_1_STA_0.M707 )
      I_Contact( "DB347_M_UNIT_1_STA_3".M_CODES_UNIT_1_STA_3.M707 )
      I_Contact( "DB353_M_UNIT_1_STA_4".M_CODES_UNIT_1_STA_4.M707 )
      Not()
   END_RUNG wire#w2
   RUNG wire#powerrail
      Contact( "DB341_M_UNIT_1_STA_0".M_CODES_UNIT_1_STA_0.M720 )
   END_RUNG wire#w3
   RUNG wire#powerrail
      Contact( "DB341_M_UNIT_1_STA_0".M_CODES_UNIT_1_STA_0.M721 )
   END_RUNG wire#w3
   RUNG wire#powerrail
      Contact( "DB341_M_UNIT_1_STA_0".M_CODES_UNIT_1_STA_0.M722 )
   END_RUNG wire#w4
   RUNG wire#powerrail
      Contact( "DB341_M_UNIT_1_STA_0".M_CODES_UNIT_1_STA_0.M723 )
   END_RUNG wire#w4
   RUNG wire#powerrail
      I_Contact( "DB341_M_UNIT_1_STA_0".M_CODES_UNIT_1_STA_0.M50 )
      I_Contact( "DB341_M_UNIT_1_STA_0".M_CODES_UNIT_1_STA_0.M51 )
   END_RUNG wire#w5
   // the same network as SCL:
   "DB2800_UNIT_1_FIXTURE_4"(PART_PRESENT_FACE_SENSOR := "DB3000_PART_PRESENT_CONTROL_U1_STA_1".FACE_N_PART_PRESENT OR "DB3000_PART_PRESENT_CONTROL_U1_STA_1".FACE_N_MASTER_PRESENT,   // "FB2500_FIXTURE_CLADDING"
                           PART_STATUS_PRESENT := "DB8000_PART_STATUS".UNIT_1.FIXTURE_4.PART_A.STATUS.PRESENT,
                           PART_STATUS_VIRTUAL_PART := "DB8000_PART_STATUS".UNIT_1.FIXTURE_4.PART_A.STATUS.VIRTUAL_PART,
                           PART_STATUS_MASTER_PART := "DB8000_PART_STATUS".UNIT_1.FIXTURE_4.PART_A.STATUS.MASTER_PART,
                           STATION_PART_PRESENT := "DB3000_PART_PRESENT_CONTROL_U1_STA_1".PART_PRESENT_INPUT,
                           STATION_NO_PART := "DB3000_PART_PRESENT_CONTROL_U1_STA_1".NO_PART,
                           STATION_PART_HAT_POSITION := "DB3000_PART_PRESENT_CONTROL_U1_STA_1".PART_HAT_POSITION_INPUT,
                           STATION_PART_CLAMPED := "DB3001_JAW_CHUCK_CONTROL_U1_STA_1".CLAMPED,
                           STATION_PART_UNCLAMPED := "DB3001_JAW_CHUCK_CONTROL_U1_STA_1".UNCLAMPED,
                           STATION_CLAMPED_WITHOUT_PART := "DB3001_JAW_CHUCK_CONTROL_U1_STA_1".CLAMPED_WITHOUT_PART,
                           VERIFY_FIXTURE_CLAMPED := NOT (NOT "DB341_M_UNIT_1_STA_0".M_CODES_UNIT_1_STA_0.M707 AND NOT "DB347_M_UNIT_1_STA_3".M_CODES_UNIT_1_STA_3.M707 AND NOT "DB353_M_UNIT_1_STA_4".M_CODES_UNIT_1_STA_4.M707),
                           GRIPPER_CLOSE := "DB2810_U1_F4_GRIPPER".CLOSE,
                           GRIPPER_OPEN := "DB2810_U1_F4_GRIPPER".OPEN_ACTION,
                           GRIPPER_CLOSED := "DB2810_U1_F4_GRIPPER".CLOSED,
                           "GRIPPER OPENED" := "DB2810_U1_F4_GRIPPER".OPEN_STATUS,
                           M_FIXTURE_GRIPPER_CLOSE := "DB341_M_UNIT_1_STA_0".M_CODES_UNIT_1_STA_0.M720 OR "DB341_M_UNIT_1_STA_0".M_CODES_UNIT_1_STA_0.M721,
                           M_FIXTURE_GRIPPER_OPEN := "DB341_M_UNIT_1_STA_0".M_CODES_UNIT_1_STA_0.M722 OR "DB341_M_UNIT_1_STA_0".M_CODES_UNIT_1_STA_0.M723,
                           UP_SEALING_STRUCTURE_CLOSED := "DB6600_UNIT_1_UP_SEALING_STRUCTURE".CLOSED,
                           DOWN_SEALING_STRUCTURE_CLOSED := "DB6601_UNIT_1_DOWN_SEALING_STRUCTURE".CLOSED,
                           PART_TYPE_FIXTURES := "DB7215_PART_TYPE".PART_TYPE_U01_FIXTURES,
                           ROBOT_PART_LOAD_UNLOAD := NOT "DB341_M_UNIT_1_STA_0".M_CODES_UNIT_1_STA_0.M50 AND NOT "DB341_M_UNIT_1_STA_0".M_CODES_UNIT_1_STA_0.M51,
                           ROBOT_OUT_OF_COLLISION := "DB7300_INTERLOCK_GENERAL".GENERAL_MACHINE.FROM_ROBOT_TO_UNIT_1.OUT_OF_COLLISION_MACHINE,
                           E_AXIS_HOME_POS := "DB5000_FIX_TABLE_POSITIONS".UNIT_1.AXIS_E10_HOME_POS,
                           W_AXIS_CLAMP_CHECK_POS := "DB140_CLADDING_AXIS_W11".SAFETY_POSITIONS.SAFETY_POSITION_4.IN_POSITION,
                           W_AXIS_UNCLAMP_CHECK_POS := "DB140_CLADDING_AXIS_W11".SAFETY_POSITIONS.SAFETY_POSITION_2.IN_POSITION,
                           UNIT_NO := 1,
                           FIXTURE_NO := 4,
                           NOT_CLAMPED_DURING_MACHINING_A => "DB426_ALARMS_WARNINGS".ALARMS.UNIT_01."716035",
                           PART_PRESENT_DISCORDANCY_A => "DB426_ALARMS_WARNINGS".ALARMS.UNIT_01."716011",
                           PART_TYPE_DISCORDANCY_A => "DB426_ALARMS_WARNINGS".ALARMS.UNIT_01."716003",
                           PART_TYPE_ORIENTATED_DISCORDANCY_A => "DB426_ALARMS_WARNINGS".ALARMS.UNIT_01."716027");
END_REGION

REGION Network 5: CALL FC2510 GRIPPERS
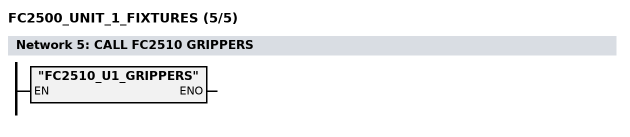
   RUNG wire#powerrail
      "FC2510_U1_GRIPPERS"()
   END_RUNG
   // the same network as SCL:
   "FC2510_U1_GRIPPERS"();
END_REGION
END_FUNCTION
